// TIA Portal project "V15_PowerDistribution" (V15)

(* hardware
DEVICE "S7-1200 station_2"  S7-1200 Station
   slot 0: "Rack_0"  S7-1200 Rack  Rack  V1.0
   slot 1: "Main_PLC"  CPU 1214C DC/DC/DC  6ES7 214-1AG31-0XB0  V3.0
DEVICE "Main_HMI"  KTP700 Basic PN
   slot 0: "Main_HMI"  KTP700 Basic PN  6AV2 123-2GB03-0AX0  15.0.0.0
   slot 1: "HMI_RT_2"  KTP700 Basic PN  6AV2 123-2GB03-0AX0  15.0.0.0
   slot 5: "Main_HMI.IE_CP_1"  PROFINET Interface  15.0.0.0
      slot 1: "PROFINET Interface_1"  PROFINET Interface
         slot 1: "Port_1"  Port
DEVICE "S7-1200 station_1"  S7-1200 Station
   slot 0: "Rack_0"  S7-1200 Rack  Rack  V1.0
   slot 1: "Test_PLC"  CPU 1214C DC/DC/DC  6ES7 214-1AG40-0XB0  V4.2
DEVICE "Test_HMI"  KTP700 Basic PN
   slot 0: "Test_HMI"  KTP700 Basic PN  6AV2 123-2GB03-0AX0  15.0.0.0
   slot 1: "HMI_RT_1"  KTP700 Basic PN  6AV2 123-2GB03-0AX0  15.0.0.0
   slot 5: "Test_HMI.IE_CP_1"  PROFINET Interface  15.0.0.0
      slot 1: "PROFINET Interface_1"  PROFINET Interface
         slot 1: "Port_1"  Port
DEVICE "Main_PC"  SIMATIC PC station
   slot 0: "SIMATIC PC station"  Rail  SIMATIC PC-Station  V1.0
      slot 125: "Stationmanager"  Station_Manager  V6.0.4
   slot 1: "PC_HMI"  WinCC RT Advanced  6AV2 104-0xxxx-xxxx  15.0.0.0
      slot 33792: "Host interface"  Host interface
   slot 2: "IE general_1"  IE General  IE_CP  V8.2.0
*)

// ===== PLC "Main_PLC"  CPU 1214C DC/DC/DC =====

VAR_GLOBAL   // PLC tag table "Default tag table"
   "Clock_Byte" AT %MB0 : Byte;
   "Clock_10Hz" AT %M0.0 : Bool;
   "Clock_5Hz" AT %M0.1 : Bool;
   "Clock_2.5Hz" AT %M0.2 : Bool;
   "Clock_2Hz" AT %M0.3 : Bool;
   "Clock_1.25Hz" AT %M0.4 : Bool;
   "Clock_1Hz" AT %M0.5 : Bool;
   "Clock_0.625Hz" AT %M0.6 : Bool;
   "Clock_0.5Hz" AT %M0.7 : Bool;
   "Normal" AT %Q0.0 : Bool;
   "Low_Volt" AT %Q0.1 : Bool;
   "Short_Circuit" AT %Q0.2 : Bool;
   "Freq_Fault" AT %Q0.3 : Bool;
   "Open_Circuit" AT %Q0.4 : Bool;
   "Overload" AT %Q0.5 : Bool;
   "illegal_load" AT %Q0.6 : Bool;
   "Poor_PF" AT %Q0.7 : Bool;
   "CB" AT %Q1.1 : Bool;
   "Switch_auto" AT %M2.1 : Bool;
   "Switch_manual" AT %M1.0 : Bool;
   "Timer0_enable" AT %M1.1 : Bool;
END_VAR

VAR_GLOBAL   // PLC tag table "HOLD_REG"
   "Send_Frequency" AT %MW100 : Word;   // Send_Frequency
   "Send_Voltage" AT %MW102 : Word;   // Send_Voltage
   "Send_Current" AT %MW104 : Word;   // Send_Current
   "Send_EnergyHighByte" AT %MW106 : Word;   // Send_EnergyHighByte
   "Send_EnergyLowByte" AT %MW108 : Word;   // Send_EnergyLowByte
   "Send_ActivePower" AT %MW110 : Word;   // Send_ActivePower
   "Send_ReactivePower" AT %MW112 : Word;   // Send_ReactivePower
   "Send_PowerFactor" AT %MW114 : Word;   // Send_PowerFactor
   "Send_ActiveCounter" AT %MW118 : Word;   // Send_ActiveCounter
   "Recv_Frequency" AT %MW120 : Word;   // Recv_Frequency
   "Recv_Voltage" AT %MW122 : Word;   // Recv_Voltage
   "Recv_Current" AT %MW124 : Word;   // Recv_Current
   "Recv_EnergyHighByte" AT %MW126 : Word;   // Recv_EnergyHighByte
   "Recv_EnergyLowByte" AT %MW128 : Word;   // Recv_EnergyLowByte
   "Recv_ActivePower" AT %MW130 : Word;   // Recv_ActivePower
   "Recv_ReactivePower" AT %MW132 : Word;   // Recv_ReactivePower
   "Recv_PowerFactor" AT %MW134 : Word;   // Recv_PowerFactor
   "Recv_ErrorFlag" AT %MW136 : Word;   // Recv_ErrorFlag
   "Recv_ActiveCounter" AT %MW138 : Word;   // Recv_ActiveCounter
   "Send_ErrorFlag" AT %MW116 : Word;   // Send_ErrorFlag
END_VAR

DATA_BLOCK "Input_DB"   // DB1
{ S7_Optimized_Access := 'TRUE' }
VERSION : 0.1
   VAR
      "Send_Frequency [Hz]" : DInt := 0;
      "Send_Voltage [V]" : DInt := 0;
      "Send_Current [A]" : DInt := 0;
      "Send_Energy [KWh]" : DInt;
      "Send_ActivePwr [W]" : DInt := 0;
      "Send_ReactivePwr [KVAr]" : DInt;
      Send_PwrFactor : DInt := 0;
      "Recv_Frequency [Hz]" : DInt := 0;
      "Recv_Voltage [V]" : DInt := 0;
      "Recv_Current [A]" : DInt := 0;
      "Recv_Energy [KWh]" : DInt;
      "Recv_ActivePwr [W]" : DInt := 0;
      "Recv_ReactivePwr [KVAr]" : DInt;
      Recv_PwrFactor : DInt := 0;
      Send_Error : DInt;
      Recv_Error : DInt;
      Send_ActiveCounter : DInt;
      Recv_ActiveCounter : DInt;
   END_VAR
BEGIN
END_DATA_BLOCK

DATA_BLOCK "MB_Server_Data"   // DB2
{ S7_Optimized_Access := 'TRUE' }
VERSION : 0.1
   VAR
      CONNECT_ID : UInt := 2;
      IP_PORT : UInt := 502;
      NDR : Bool;
      DR : Bool;
      ERROR : Bool;
      STATUS : Word;
   END_VAR
BEGIN
END_DATA_BLOCK

DATA_BLOCK "Cond_DB"   // DB3
{ S7_Optimized_Access := 'TRUE' }
VERSION : 0.1
   VAR
      Recv_PwrLimit : DInt := 1000;
      error_ActivePwr : DInt;
      Psend_10percent : DInt;
      PwrFactor_Limit : DInt := 500;
      Freq_LowerLImit : DInt := 4750;
      Freq_UpperLimit : DInt := 5250;
      Current_Limit : DInt := 2;
      Vsend_limit_5percent : DInt := 2200;
      Vsend_limit_10percent : DInt := 2080;
      Vsend_High : DInt := 2420;
   END_VAR
BEGIN
END_DATA_BLOCK

DATA_BLOCK "MB_Client_Data"   // DB5
{ S7_Optimized_Access := 'TRUE' }
VERSION : 0.1
   VAR
      DISCONNECT : Bool;
      CONNECT_ID : UInt := 1;
      IP_ADDRESS : Array[0..3] of Byte;
      IP_PORT : UInt := 502;
      MB_MODE : USInt := 1;
      DATA_ADDRESS : UDInt := 0;
      DATA_LEN : UInt := 20;
      DONE : Bool;
      BUSY : Bool;
      ERROR : Bool;
      STATUS : Word;
   END_VAR
BEGIN
   IP_ADDRESS[0] := 192;
   IP_ADDRESS[1] := 168;
   IP_ADDRESS[2] := 0;
   IP_ADDRESS[3] := 103;
END_DATA_BLOCK

DATA_BLOCK "Fault_DB"   // DB6
{ S7_Optimized_Access := 'TRUE' }
VERSION : 0.1
   VAR
      None : Bool;
      Low_Voltage : Bool;
      Short_Circuit : Bool;
      Freq_fault : Bool;
      Open_Circuit : Bool;
      High_Voltage : Bool;
      Overload : Bool;
      Illegal_Load : Bool;
      Poor_PF : Bool;
   END_VAR
BEGIN
END_DATA_BLOCK

// folder: System blocks/Program resources

DATA_BLOCK "IEC_Timer_0_DB"   // DB7
{ S7_Optimized_Access := 'TRUE' }
AUTHOR : Simatic
FAMILY : IEC
NAME : IEC_TMR
VERSION : 1.0
// stored: InstanceOfName IEC_TIMER
"IEC_TIMER"
BEGIN
END_DATA_BLOCK

DATA_BLOCK "IEC_Timer_0_DB_1"   // DB9
{ S7_Optimized_Access := 'TRUE' }
AUTHOR : Simatic
FAMILY : IEC
NAME : IEC_TMR
VERSION : 1.0
// stored: InstanceOfName IEC_TIMER
"IEC_TIMER"
BEGIN
END_DATA_BLOCK

DATA_BLOCK "IEC_Timer_0_DB_2"   // DB10
{ S7_Optimized_Access := 'TRUE' }
AUTHOR : Simatic
FAMILY : IEC
NAME : IEC_TMR
VERSION : 1.0
// stored: InstanceOfName IEC_TIMER
"IEC_TIMER"
BEGIN
END_DATA_BLOCK

DATA_BLOCK "IEC_Timer_0_DB_3"   // DB11
{ S7_Optimized_Access := 'TRUE' }
AUTHOR : Simatic
FAMILY : IEC
NAME : IEC_TMR
VERSION : 1.0
// stored: InstanceOfName IEC_TIMER
"IEC_TIMER"
BEGIN
END_DATA_BLOCK

// folder: (top level)

ORGANIZATION_BLOCK "Main"   // OB1, LAD, ProgramCycle
TITLE = "Main Program Sweep (Cycle)"
{ S7_Optimized_Access := 'TRUE' }
VERSION : 0.1
   VAR_INPUT
      Initial_Call : Bool;   // Initial call of this OB
      Remanence : Bool;   // =True, if remanent data are available
   END_VAR
   VAR_TEMP
      Freq_Fault : Bool;
   END_VAR
BEGIN

REGION Network 1: Detect Fault
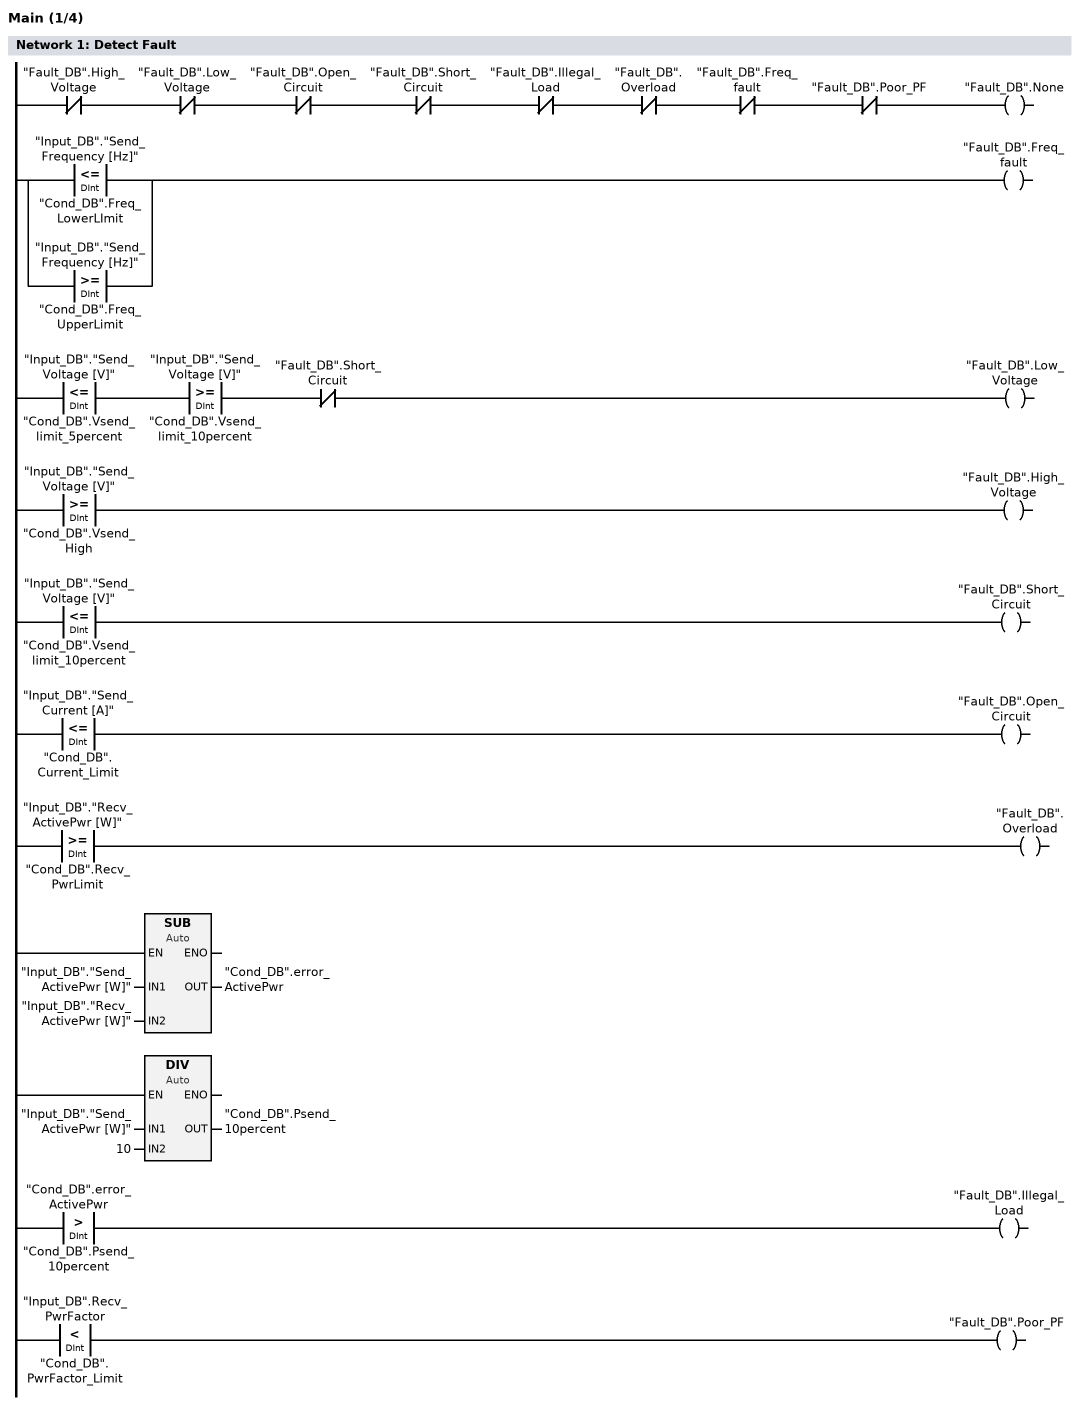
   RUNG wire#powerrail
      I_Contact( "Fault_DB".High_Voltage )
      I_Contact( "Fault_DB".Low_Voltage )
      I_Contact( "Fault_DB".Open_Circuit )
      I_Contact( "Fault_DB".Short_Circuit )
      I_Contact( "Fault_DB".Illegal_Load )
      I_Contact( "Fault_DB".Overload )
      I_Contact( "Fault_DB".Freq_fault )
      I_Contact( "Fault_DB".Poor_PF )
      Coil( "Fault_DB".None )
   END_RUNG
   RUNG wire#powerrail
      { S7_Templates := "SrcType := DInt" } LE_Contact(in1 := "Input_DB"."Send_Frequency [Hz]", in2 := "Cond_DB".Freq_LowerLImit)
      wire#w1
      Coil( "Fault_DB".Freq_fault )
   END_RUNG
   RUNG wire#powerrail
      { S7_Templates := "SrcType := DInt" } GE_Contact(in1 := "Input_DB"."Send_Frequency [Hz]", in2 := "Cond_DB".Freq_UpperLimit)
   END_RUNG wire#w1
   RUNG wire#powerrail
      { S7_Templates := "SrcType := DInt" } LE_Contact(in1 := "Input_DB"."Send_Voltage [V]", in2 := "Cond_DB".Vsend_limit_5percent)
      { S7_Templates := "SrcType := DInt" } GE_Contact(in1 := "Input_DB"."Send_Voltage [V]", in2 := "Cond_DB".Vsend_limit_10percent)
      I_Contact( "Fault_DB".Short_Circuit )
      Coil( "Fault_DB".Low_Voltage )
   END_RUNG
   RUNG wire#powerrail
      { S7_Templates := "SrcType := DInt" } GE_Contact(in1 := "Input_DB"."Send_Voltage [V]", in2 := "Cond_DB".Vsend_High)
      Coil( "Fault_DB".High_Voltage )
   END_RUNG
   RUNG wire#powerrail
      { S7_Templates := "SrcType := DInt" } LE_Contact(in1 := "Input_DB"."Send_Voltage [V]", in2 := "Cond_DB".Vsend_limit_10percent)
      Coil( "Fault_DB".Short_Circuit )
   END_RUNG
   RUNG wire#powerrail
      { S7_Templates := "SrcType := DInt" } LE_Contact(in1 := "Input_DB"."Send_Current [A]", in2 := "Cond_DB".Current_Limit)
      Coil( "Fault_DB".Open_Circuit )
   END_RUNG
   RUNG wire#powerrail
      { S7_Templates := "SrcType := DInt" } GE_Contact(in1 := "Input_DB"."Recv_ActivePwr [W]", in2 := "Cond_DB".Recv_PwrLimit)
      Coil( "Fault_DB".Overload )
   END_RUNG
   RUNG wire#powerrail
      { S7_GenerateENO := "TRUE" } Sub(in1 := "Input_DB"."Send_ActivePwr [W]", in2 := "Input_DB"."Recv_ActivePwr [W]", out => "Cond_DB".error_ActivePwr)
   END_RUNG
   RUNG wire#powerrail
      { S7_GenerateENO := "TRUE" } Div(in1 := "Input_DB"."Send_ActivePwr [W]", in2 := 10, out => "Cond_DB".Psend_10percent)
   END_RUNG
   RUNG wire#powerrail
      { S7_Templates := "SrcType := DInt" } GT_Contact(in1 := "Cond_DB".error_ActivePwr, in2 := "Cond_DB".Psend_10percent)
      Coil( "Fault_DB".Illegal_Load )
   END_RUNG
   RUNG wire#powerrail
      { S7_Templates := "SrcType := DInt" } LT_Contact(in1 := "Input_DB".Recv_PwrFactor, in2 := "Cond_DB".PwrFactor_Limit)
      Coil( "Fault_DB".Poor_PF )
   END_RUNG
   // the same network as SCL:
   "Fault_DB".None := NOT "Fault_DB".High_Voltage AND NOT "Fault_DB".Low_Voltage AND NOT "Fault_DB".Open_Circuit AND NOT "Fault_DB".Short_Circuit AND NOT "Fault_DB".Illegal_Load AND NOT "Fault_DB".Overload AND NOT "Fault_DB".Freq_fault AND NOT "Fault_DB".Poor_PF;
   "Fault_DB".Freq_fault := ("Input_DB"."Send_Frequency [Hz]" <= "Cond_DB".Freq_LowerLImit) OR ("Input_DB"."Send_Frequency [Hz]" >= "Cond_DB".Freq_UpperLimit);
   "Fault_DB".Low_Voltage := ("Input_DB"."Send_Voltage [V]" <= "Cond_DB".Vsend_limit_5percent) AND ("Input_DB"."Send_Voltage [V]" >= "Cond_DB".Vsend_limit_10percent) AND NOT "Fault_DB".Short_Circuit;
   "Fault_DB".High_Voltage := "Input_DB"."Send_Voltage [V]" >= "Cond_DB".Vsend_High;
   "Fault_DB".Short_Circuit := "Input_DB"."Send_Voltage [V]" <= "Cond_DB".Vsend_limit_10percent;
   "Fault_DB".Open_Circuit := "Input_DB"."Send_Current [A]" <= "Cond_DB".Current_Limit;
   "Fault_DB".Overload := "Input_DB"."Recv_ActivePwr [W]" >= "Cond_DB".Recv_PwrLimit;
   "Cond_DB".error_ActivePwr := "Input_DB"."Send_ActivePwr [W]" - "Input_DB"."Recv_ActivePwr [W]";
   "Cond_DB".Psend_10percent := "Input_DB"."Send_ActivePwr [W]" / 10;
   "Fault_DB".Illegal_Load := "Cond_DB".error_ActivePwr > "Cond_DB".Psend_10percent;
   "Fault_DB".Poor_PF := "Input_DB".Recv_PwrFactor < "Cond_DB".PwrFactor_Limit;
END_REGION

REGION Network 2: Display Fault
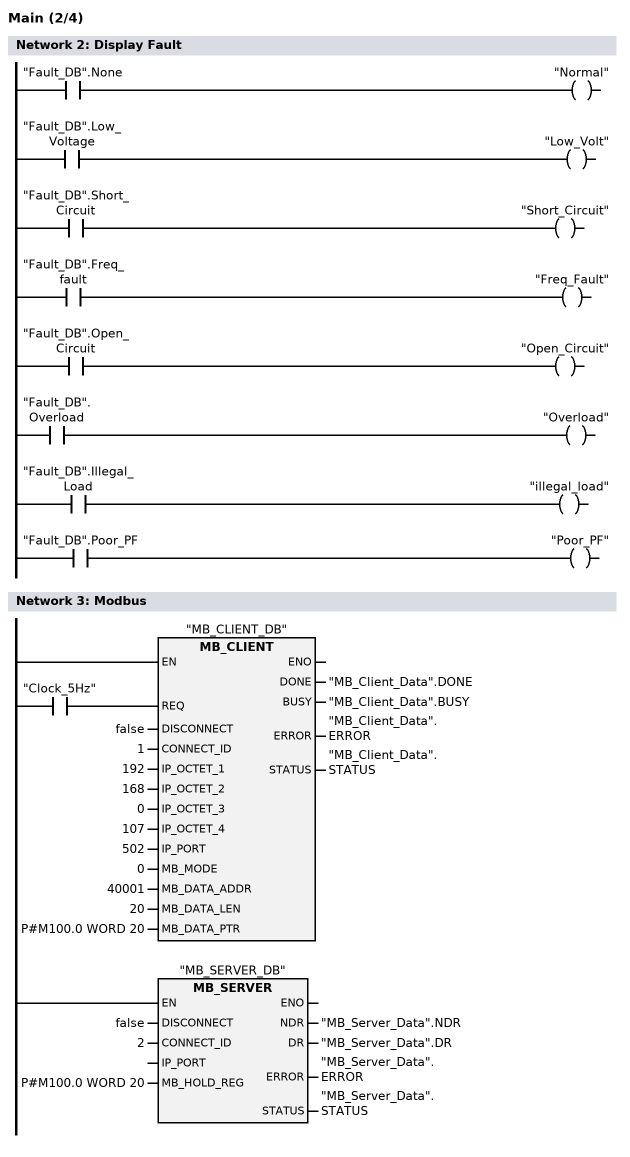
   RUNG wire#powerrail
      Contact( "Fault_DB".None )
      Coil( "Normal" )
   END_RUNG
   RUNG wire#powerrail
      Contact( "Fault_DB".Low_Voltage )
      Coil( "Low_Volt" )
   END_RUNG
   RUNG wire#powerrail
      Contact( "Fault_DB".Short_Circuit )
      Coil( "Short_Circuit" )
   END_RUNG
   RUNG wire#powerrail
      Contact( "Fault_DB".Freq_fault )
      Coil( "Freq_Fault" )
   END_RUNG
   RUNG wire#powerrail
      Contact( "Fault_DB".Open_Circuit )
      Coil( "Open_Circuit" )
   END_RUNG
   RUNG wire#powerrail
      Contact( "Fault_DB".Overload )
      Coil( "Overload" )
   END_RUNG
   RUNG wire#powerrail
      Contact( "Fault_DB".Illegal_Load )
      Coil( "illegal_load" )
   END_RUNG
   RUNG wire#powerrail
      Contact( "Fault_DB".Poor_PF )
      Coil( "Poor_PF" )
   END_RUNG
   // the same network as SCL:
   "Normal" := "Fault_DB".None;
   "Low_Volt" := "Fault_DB".Low_Voltage;
   "Short_Circuit" := "Fault_DB".Short_Circuit;
   "Freq_Fault" := "Fault_DB".Freq_fault;
   "Open_Circuit" := "Fault_DB".Open_Circuit;
   "Overload" := "Fault_DB".Overload;
   "illegal_load" := "Fault_DB".Illegal_Load;
   "Poor_PF" := "Fault_DB".Poor_PF;
END_REGION

REGION Network 3: Modbus
   "MB_CLIENT_DB"(REQ := "Clock_5Hz",   // MB_CLIENT
                  DISCONNECT := false,
                  CONNECT_ID := 1,
                  IP_OCTET_1 := 192,
                  IP_OCTET_2 := 168,
                  IP_OCTET_3 := 0,
                  IP_OCTET_4 := 107,
                  IP_PORT := 502,
                  MB_MODE := 0,
                  MB_DATA_ADDR := 40001,
                  MB_DATA_LEN := 20,
                  MB_DATA_PTR := P#M100.0 WORD 20,
                  DONE => "MB_Client_Data".DONE,
                  BUSY => "MB_Client_Data".BUSY,
                  ERROR => "MB_Client_Data".ERROR,
                  STATUS => "MB_Client_Data".STATUS);
   "MB_SERVER_DB"(DISCONNECT := false,   // MB_SERVER
                  CONNECT_ID := 2,
                  MB_HOLD_REG := P#M100.0 WORD 20,
                  NDR => "MB_Server_Data".NDR,
                  DR => "MB_Server_Data".DR,
                  ERROR => "MB_Server_Data".ERROR,
                  STATUS => "MB_Server_Data".STATUS);
END_REGION

REGION Network 4: Map data from sensors to DB
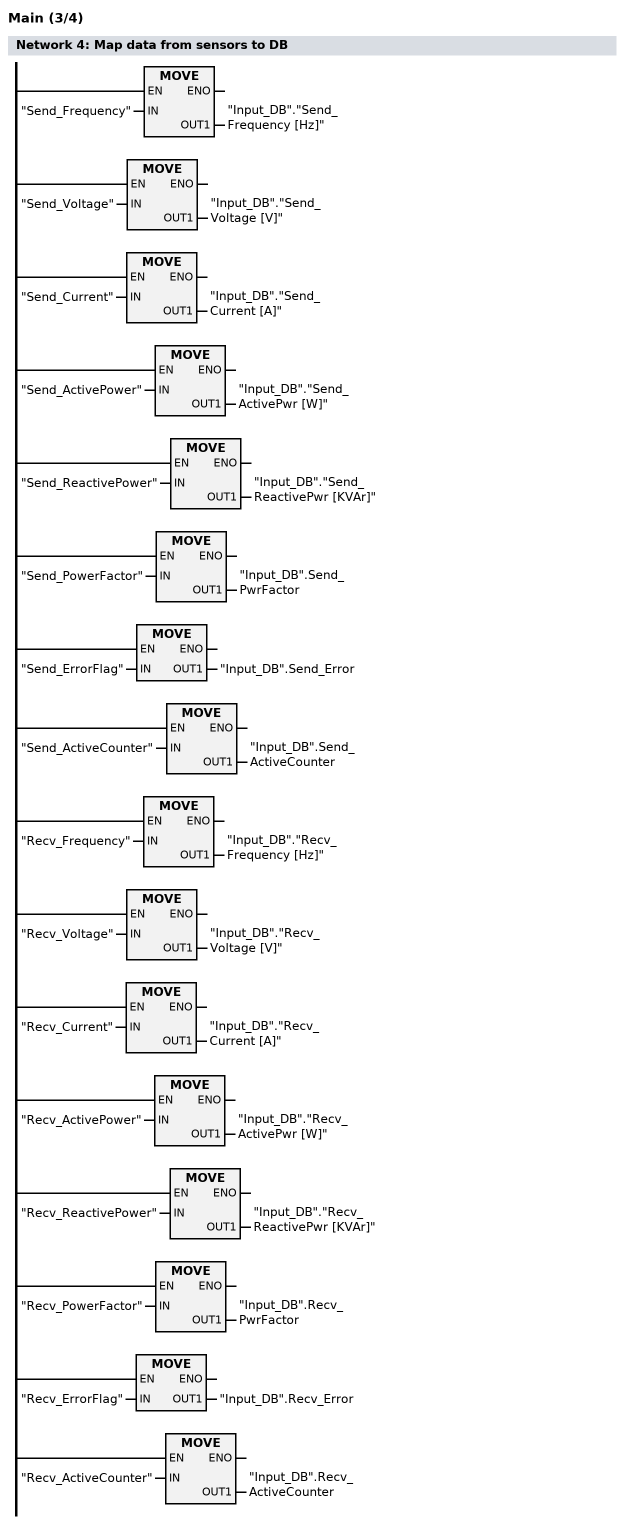
   RUNG wire#powerrail
      { S7_GenerateENO := "TRUE" } Move(in := "Send_Frequency", out1 => "Input_DB"."Send_Frequency [Hz]")
   END_RUNG
   RUNG wire#powerrail
      { S7_GenerateENO := "TRUE" } Move(in := "Send_Voltage", out1 => "Input_DB"."Send_Voltage [V]")
   END_RUNG
   RUNG wire#powerrail
      { S7_GenerateENO := "TRUE" } Move(in := "Send_Current", out1 => "Input_DB"."Send_Current [A]")
   END_RUNG
   RUNG wire#powerrail
      { S7_GenerateENO := "TRUE" } Move(in := "Send_ActivePower", out1 => "Input_DB"."Send_ActivePwr [W]")
   END_RUNG
   RUNG wire#powerrail
      { S7_GenerateENO := "TRUE" } Move(in := "Send_ReactivePower", out1 => "Input_DB"."Send_ReactivePwr [KVAr]")
   END_RUNG
   RUNG wire#powerrail
      { S7_GenerateENO := "TRUE" } Move(in := "Send_PowerFactor", out1 => "Input_DB".Send_PwrFactor)
   END_RUNG
   RUNG wire#powerrail
      { S7_GenerateENO := "TRUE" } Move(in := "Send_ErrorFlag", out1 => "Input_DB".Send_Error)
   END_RUNG
   RUNG wire#powerrail
      { S7_GenerateENO := "TRUE" } Move(in := "Send_ActiveCounter", out1 => "Input_DB".Send_ActiveCounter)
   END_RUNG
   RUNG wire#powerrail
      { S7_GenerateENO := "TRUE" } Move(in := "Recv_Frequency", out1 => "Input_DB"."Recv_Frequency [Hz]")
   END_RUNG
   RUNG wire#powerrail
      { S7_GenerateENO := "TRUE" } Move(in := "Recv_Voltage", out1 => "Input_DB"."Recv_Voltage [V]")
   END_RUNG
   RUNG wire#powerrail
      { S7_GenerateENO := "TRUE" } Move(in := "Recv_Current", out1 => "Input_DB"."Recv_Current [A]")
   END_RUNG
   RUNG wire#powerrail
      { S7_GenerateENO := "TRUE" } Move(in := "Recv_ActivePower", out1 => "Input_DB"."Recv_ActivePwr [W]")
   END_RUNG
   RUNG wire#powerrail
      { S7_GenerateENO := "TRUE" } Move(in := "Recv_ReactivePower", out1 => "Input_DB"."Recv_ReactivePwr [KVAr]")
   END_RUNG
   RUNG wire#powerrail
      { S7_GenerateENO := "TRUE" } Move(in := "Recv_PowerFactor", out1 => "Input_DB".Recv_PwrFactor)
   END_RUNG
   RUNG wire#powerrail
      { S7_GenerateENO := "TRUE" } Move(in := "Recv_ErrorFlag", out1 => "Input_DB".Recv_Error)
   END_RUNG
   RUNG wire#powerrail
      { S7_GenerateENO := "TRUE" } Move(in := "Recv_ActiveCounter", out1 => "Input_DB".Recv_ActiveCounter)
   END_RUNG
   // the same network as SCL:
   "Input_DB"."Send_Frequency [Hz]" := "Send_Frequency";
   "Input_DB"."Send_Voltage [V]" := "Send_Voltage";
   "Input_DB"."Send_Current [A]" := "Send_Current";
   "Input_DB"."Send_ActivePwr [W]" := "Send_ActivePower";
   "Input_DB"."Send_ReactivePwr [KVAr]" := "Send_ReactivePower";
   "Input_DB".Send_PwrFactor := "Send_PowerFactor";
   "Input_DB".Send_Error := "Send_ErrorFlag";
   "Input_DB".Send_ActiveCounter := "Send_ActiveCounter";
   "Input_DB"."Recv_Frequency [Hz]" := "Recv_Frequency";
   "Input_DB"."Recv_Voltage [V]" := "Recv_Voltage";
   "Input_DB"."Recv_Current [A]" := "Recv_Current";
   "Input_DB"."Recv_ActivePwr [W]" := "Recv_ActivePower";
   "Input_DB"."Recv_ReactivePwr [KVAr]" := "Recv_ReactivePower";
   "Input_DB".Recv_PwrFactor := "Recv_PowerFactor";
   "Input_DB".Recv_Error := "Recv_ErrorFlag";
   "Input_DB".Recv_ActiveCounter := "Recv_ActiveCounter";
END_REGION

REGION Network 5: Circuit Breaker Switch
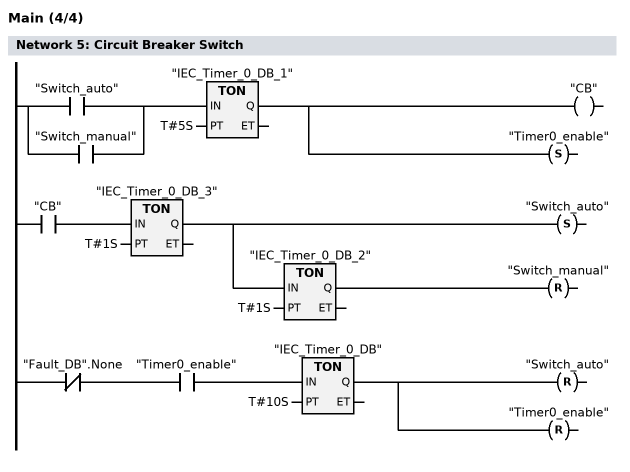
   "IEC_Timer_0_DB_1".TON(IN := "Switch_auto" OR "Switch_manual", PT := T#5S);
   "CB" := "IEC_Timer_0_DB_1".Q;
   IF "IEC_Timer_0_DB_1".Q THEN "Timer0_enable" := TRUE; END_IF;
   "IEC_Timer_0_DB_3".TON(IN := "CB", PT := T#1S);
   IF "IEC_Timer_0_DB_3".Q THEN "Switch_auto" := TRUE; END_IF;
   "IEC_Timer_0_DB_2".TON(IN := "IEC_Timer_0_DB_3".Q, PT := T#1S);
   IF "IEC_Timer_0_DB_2".Q THEN "Switch_manual" := FALSE; END_IF;
   "IEC_Timer_0_DB".TON(IN := NOT "Fault_DB".None AND "Timer0_enable", PT := T#10S);
   IF "IEC_Timer_0_DB".Q THEN
       "Switch_auto" := FALSE;
       "Timer0_enable" := FALSE;
   END_IF;
END_REGION
END_ORGANIZATION_BLOCK

// ===== PLC "Test_PLC"  CPU 1214C DC/DC/DC =====

VAR_GLOBAL   // PLC tag table "Default tag table"
   "Clock_Byte" AT %MB0 : Byte;
   "Clock_10Hz" AT %M0.0 : Bool;
   "Clock_5Hz" AT %M0.1 : Bool;
   "Clock_2.5Hz" AT %M0.2 : Bool;
   "Clock_2Hz" AT %M0.3 : Bool;
   "Clock_1.25Hz" AT %M0.4 : Bool;
   "Clock_1Hz" AT %M0.5 : Bool;
   "Clock_0.625Hz" AT %M0.6 : Bool;
   "Clock_0.5Hz" AT %M0.7 : Bool;
   "Normal" AT %M1.0 : Bool;
   "Low_Volt" AT %M1.1 : Bool;
   "Short_Circuit" AT %M1.2 : Bool;
   "Freq_Fault" AT %M1.3 : Bool;
   "Open_Circuit" AT %M1.4 : Bool;
   "Overload" AT %M1.5 : Bool;
   "illegal_load" AT %M1.6 : Bool;
   "Poor_PF" AT %M1.7 : Bool;
   "CB" AT %M2.0 : Bool;
   "CB_enable" AT %M2.1 : Bool;
END_VAR

VAR_GLOBAL   // PLC tag table "HOLD_REG"
   "40001" AT %MW100 : Word;   // Send_Frequency
   "40002" AT %MW102 : Word;   // Send_Voltage
   "40003" AT %MW104 : Word;   // Send_Current
   "40004" AT %MW106 : Word;   // Send_EnergyHighByte
   "40005" AT %MW108 : Word;   // Send_EnergyLowByte
   "40006" AT %MW110 : Word;   // Send_ActivePower
   "40007" AT %MW112 : Word;   // Send_ReactivePower
   "40008" AT %MW114 : Word;   // Send_PowerFactor
   "40009" AT %MW116 : Word;   // Recv_Frequency
   "40010" AT %MW118 : Word;   // Recv_Voltage
   "40011" AT %MW120 : Word;   // Recv_Current
   "40012" AT %MW122 : Word;   // Recv_EnergyHighByte
   "40013" AT %MW124 : Word;   // Recv_EnergyLowByte
   "40014" AT %MW126 : Word;   // Recv_ActivePower
   "40015" AT %MW128 : Word;   // Recv_ReactivePower
   "40016" AT %MW130 : Word;   // Recv_PowerFactor
   "40017" AT %MW132 : Word;   // Send_ErrorFlag
   "40018" AT %MW134 : Word;   // Recv_ErrorFlag
   "40019" AT %MW136 : Word;   // Send_ActiveCounter
   "40020" AT %MW138 : Word;   // Recv_ActiveCounter
END_VAR

DATA_BLOCK "Input_DB"   // DB1
{ S7_Optimized_Access := 'TRUE' }
VERSION : 0.1
   VAR
      "Send_Frequency [Hz]" : DInt := 0;
      "Send_Voltage [V]" : DInt := 0;
      "Send_Current [mA]" : DInt := 0;
      "Send_Energy [KWh]" : DInt;
      "Send_ActivePwr [W]" : DInt := 0;
      "Send_ReactivePwr [KVAr]" : DInt;
      Send_PwrFactor : DInt := 0;
      "Recv_Frequency [Hz]" : DInt := 0;
      "Recv_Voltage [V]" : DInt := 0;
      "Recv_Current [mA]" : DInt := 0;
      "Recv_Energy [KWh]" : DInt;
      "Recv_ActivePwr [W]" : DInt := 0;
      "Recv_ReactivePwr [KVAr]" : DInt;
      Recv_PwrFactor : DInt := 0;
      Send_Error : DInt;
      Recv_Error : DInt;
      Send_ActiveCounter : DInt;
      Recv_ActiveCounter : DInt;
   END_VAR
BEGIN
END_DATA_BLOCK

DATA_BLOCK "Fault_DB"   // DB2
{ S7_Optimized_Access := 'TRUE' }
VERSION : 0.1
   VAR
      None : Bool;
      Low_Voltage : Bool;
      Short_Circuit : Bool;
      Freq_fault : Bool;
      Open_Circuit : Bool;
      High_Voltage : Bool;
      Overload : Bool;
      Illegal_Load : Bool;
      Poor_PF : Bool;
   END_VAR
BEGIN
END_DATA_BLOCK

DATA_BLOCK "Cond_DB"   // DB3
{ S7_Optimized_Access := 'TRUE' }
VERSION : 0.1
   VAR
      Recv_PwrLimit : DInt := 1000;
      error_ActivePwr : DInt;
      Psend_10percent : DInt;
      PwrFactor_Limit : DInt := 800;
      Freq_LowerLImit : DInt := 4750;
      Freq_UpperLimit : DInt := 5250;
      Current_Limit : DInt := 2;
      Vsend_limit_5percent : DInt := 2200;
      Vsend_limit_10percent : DInt := 2080;
      Vsend_High : DInt := 2420;
   END_VAR
BEGIN
END_DATA_BLOCK

DATA_BLOCK "MB_Client_Data"   // DB5
{ S7_Optimized_Access := 'TRUE' }
VERSION : 0.1
   VAR
      DISCONNECT : Bool;
      CONNECT_ID : UInt := 1;
      IP_ADDRESS : Array[0..3] of Byte;
      IP_PORT : UInt := 502;
      MB_MODE : USInt := 1;
      DATA_ADDRESS : UDInt := 0;
      DATA_LEN : UInt := 20;
      DONE : Bool;
      BUSY : Bool;
      ERROR : Bool;
      STATUS : Word;
   END_VAR
BEGIN
   IP_ADDRESS[0] := 192;
   IP_ADDRESS[1] := 168;
   IP_ADDRESS[2] := 0;
   IP_ADDRESS[3] := 103;
END_DATA_BLOCK

ORGANIZATION_BLOCK "Main"   // OB1, LAD, ProgramCycle
TITLE = "Main Program Sweep (Cycle)"
{ S7_Optimized_Access := 'TRUE' }
VERSION : 0.1
   VAR_INPUT
      Initial_Call : Bool;   // Initial call of this OB
      Remanence : Bool;   // =True, if remanent data are available
   END_VAR
   VAR_TEMP
      Freq_Fault : Bool;
   END_VAR
BEGIN

REGION Network 1: Detect Fault
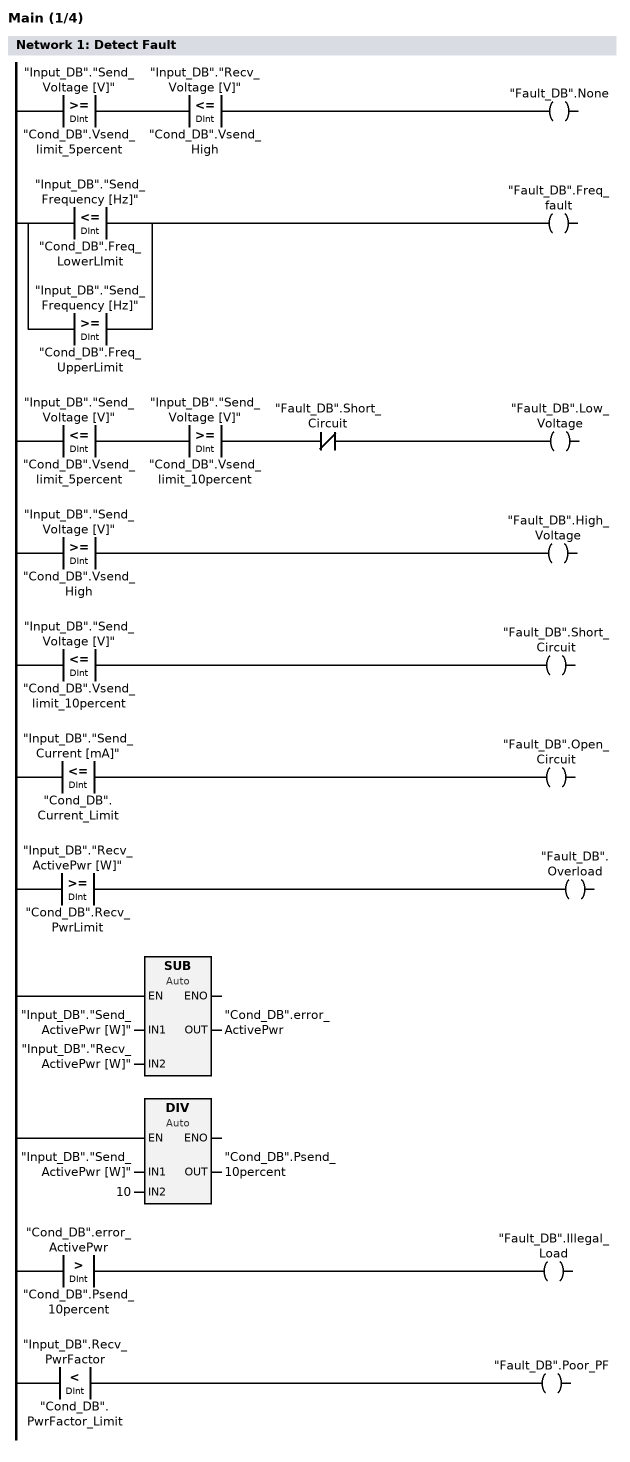
   RUNG wire#powerrail
      { S7_Templates := "SrcType := DInt" } GE_Contact(in1 := "Input_DB"."Send_Voltage [V]", in2 := "Cond_DB".Vsend_limit_5percent)
      { S7_Templates := "SrcType := DInt" } LE_Contact(in1 := "Input_DB"."Recv_Voltage [V]", in2 := "Cond_DB".Vsend_High)
      Coil( "Fault_DB".None )
   END_RUNG
   RUNG wire#powerrail
      { S7_Templates := "SrcType := DInt" } LE_Contact(in1 := "Input_DB"."Send_Frequency [Hz]", in2 := "Cond_DB".Freq_LowerLImit)
      wire#w1
      Coil( "Fault_DB".Freq_fault )
   END_RUNG
   RUNG wire#powerrail
      { S7_Templates := "SrcType := DInt" } GE_Contact(in1 := "Input_DB"."Send_Frequency [Hz]", in2 := "Cond_DB".Freq_UpperLimit)
   END_RUNG wire#w1
   RUNG wire#powerrail
      { S7_Templates := "SrcType := DInt" } LE_Contact(in1 := "Input_DB"."Send_Voltage [V]", in2 := "Cond_DB".Vsend_limit_5percent)
      { S7_Templates := "SrcType := DInt" } GE_Contact(in1 := "Input_DB"."Send_Voltage [V]", in2 := "Cond_DB".Vsend_limit_10percent)
      I_Contact( "Fault_DB".Short_Circuit )
      Coil( "Fault_DB".Low_Voltage )
   END_RUNG
   RUNG wire#powerrail
      { S7_Templates := "SrcType := DInt" } GE_Contact(in1 := "Input_DB"."Send_Voltage [V]", in2 := "Cond_DB".Vsend_High)
      Coil( "Fault_DB".High_Voltage )
   END_RUNG
   RUNG wire#powerrail
      { S7_Templates := "SrcType := DInt" } LE_Contact(in1 := "Input_DB"."Send_Voltage [V]", in2 := "Cond_DB".Vsend_limit_10percent)
      Coil( "Fault_DB".Short_Circuit )
   END_RUNG
   RUNG wire#powerrail
      { S7_Templates := "SrcType := DInt" } LE_Contact(in1 := "Input_DB"."Send_Current [mA]", in2 := "Cond_DB".Current_Limit)
      Coil( "Fault_DB".Open_Circuit )
   END_RUNG
   RUNG wire#powerrail
      { S7_Templates := "SrcType := DInt" } GE_Contact(in1 := "Input_DB"."Recv_ActivePwr [W]", in2 := "Cond_DB".Recv_PwrLimit)
      Coil( "Fault_DB".Overload )
   END_RUNG
   RUNG wire#powerrail
      { S7_GenerateENO := "TRUE" } Sub(in1 := "Input_DB"."Send_ActivePwr [W]", in2 := "Input_DB"."Recv_ActivePwr [W]", out => "Cond_DB".error_ActivePwr)
   END_RUNG
   RUNG wire#powerrail
      { S7_GenerateENO := "TRUE" } Div(in1 := "Input_DB"."Send_ActivePwr [W]", in2 := 10, out => "Cond_DB".Psend_10percent)
   END_RUNG
   RUNG wire#powerrail
      { S7_Templates := "SrcType := DInt" } GT_Contact(in1 := "Cond_DB".error_ActivePwr, in2 := "Cond_DB".Psend_10percent)
      Coil( "Fault_DB".Illegal_Load )
   END_RUNG
   RUNG wire#powerrail
      { S7_Templates := "SrcType := DInt" } LT_Contact(in1 := "Input_DB".Recv_PwrFactor, in2 := "Cond_DB".PwrFactor_Limit)
      Coil( "Fault_DB".Poor_PF )
   END_RUNG
   // the same network as SCL:
   "Fault_DB".None := ("Input_DB"."Send_Voltage [V]" >= "Cond_DB".Vsend_limit_5percent) AND ("Input_DB"."Recv_Voltage [V]" <= "Cond_DB".Vsend_High);
   "Fault_DB".Freq_fault := ("Input_DB"."Send_Frequency [Hz]" <= "Cond_DB".Freq_LowerLImit) OR ("Input_DB"."Send_Frequency [Hz]" >= "Cond_DB".Freq_UpperLimit);
   "Fault_DB".Low_Voltage := ("Input_DB"."Send_Voltage [V]" <= "Cond_DB".Vsend_limit_5percent) AND ("Input_DB"."Send_Voltage [V]" >= "Cond_DB".Vsend_limit_10percent) AND NOT "Fault_DB".Short_Circuit;
   "Fault_DB".High_Voltage := "Input_DB"."Send_Voltage [V]" >= "Cond_DB".Vsend_High;
   "Fault_DB".Short_Circuit := "Input_DB"."Send_Voltage [V]" <= "Cond_DB".Vsend_limit_10percent;
   "Fault_DB".Open_Circuit := "Input_DB"."Send_Current [mA]" <= "Cond_DB".Current_Limit;
   "Fault_DB".Overload := "Input_DB"."Recv_ActivePwr [W]" >= "Cond_DB".Recv_PwrLimit;
   "Cond_DB".error_ActivePwr := "Input_DB"."Send_ActivePwr [W]" - "Input_DB"."Recv_ActivePwr [W]";
   "Cond_DB".Psend_10percent := "Input_DB"."Send_ActivePwr [W]" / 10;
   "Fault_DB".Illegal_Load := "Cond_DB".error_ActivePwr > "Cond_DB".Psend_10percent;
   "Fault_DB".Poor_PF := "Input_DB".Recv_PwrFactor < "Cond_DB".PwrFactor_Limit;
END_REGION

REGION Network 2: Display Fault
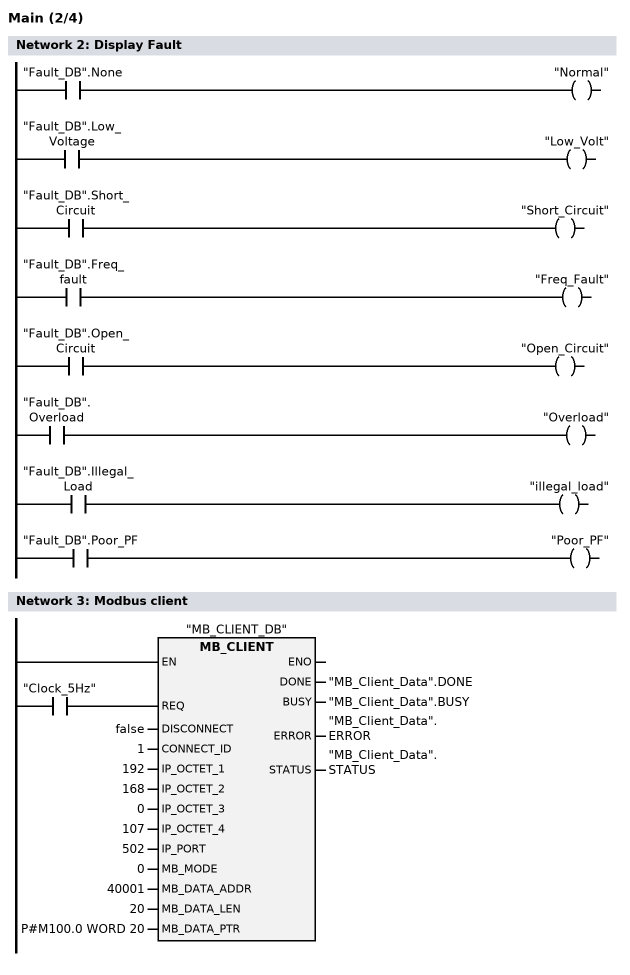
   RUNG wire#powerrail
      Contact( "Fault_DB".None )
      Coil( "Normal" )
   END_RUNG
   RUNG wire#powerrail
      Contact( "Fault_DB".Low_Voltage )
      Coil( "Low_Volt" )
   END_RUNG
   RUNG wire#powerrail
      Contact( "Fault_DB".Short_Circuit )
      Coil( "Short_Circuit" )
   END_RUNG
   RUNG wire#powerrail
      Contact( "Fault_DB".Freq_fault )
      Coil( "Freq_Fault" )
   END_RUNG
   RUNG wire#powerrail
      Contact( "Fault_DB".Open_Circuit )
      Coil( "Open_Circuit" )
   END_RUNG
   RUNG wire#powerrail
      Contact( "Fault_DB".Overload )
      Coil( "Overload" )
   END_RUNG
   RUNG wire#powerrail
      Contact( "Fault_DB".Illegal_Load )
      Coil( "illegal_load" )
   END_RUNG
   RUNG wire#powerrail
      Contact( "Fault_DB".Poor_PF )
      Coil( "Poor_PF" )
   END_RUNG
   // the same network as SCL:
   "Normal" := "Fault_DB".None;
   "Low_Volt" := "Fault_DB".Low_Voltage;
   "Short_Circuit" := "Fault_DB".Short_Circuit;
   "Freq_Fault" := "Fault_DB".Freq_fault;
   "Open_Circuit" := "Fault_DB".Open_Circuit;
   "Overload" := "Fault_DB".Overload;
   "illegal_load" := "Fault_DB".Illegal_Load;
   "Poor_PF" := "Fault_DB".Poor_PF;
END_REGION

REGION Network 3: Modbus client
   "MB_CLIENT_DB"(REQ := "Clock_5Hz",   // MB_CLIENT
                  DISCONNECT := false,
                  CONNECT_ID := 1,
                  IP_OCTET_1 := 192,
                  IP_OCTET_2 := 168,
                  IP_OCTET_3 := 0,
                  IP_OCTET_4 := 107,
                  IP_PORT := 502,
                  MB_MODE := 0,
                  MB_DATA_ADDR := 40001,
                  MB_DATA_LEN := 20,
                  MB_DATA_PTR := P#M100.0 WORD 20,
                  DONE => "MB_Client_Data".DONE,
                  BUSY => "MB_Client_Data".BUSY,
                  ERROR => "MB_Client_Data".ERROR,
                  STATUS => "MB_Client_Data".STATUS);
END_REGION

REGION Network 4: Map data from sensors to DB
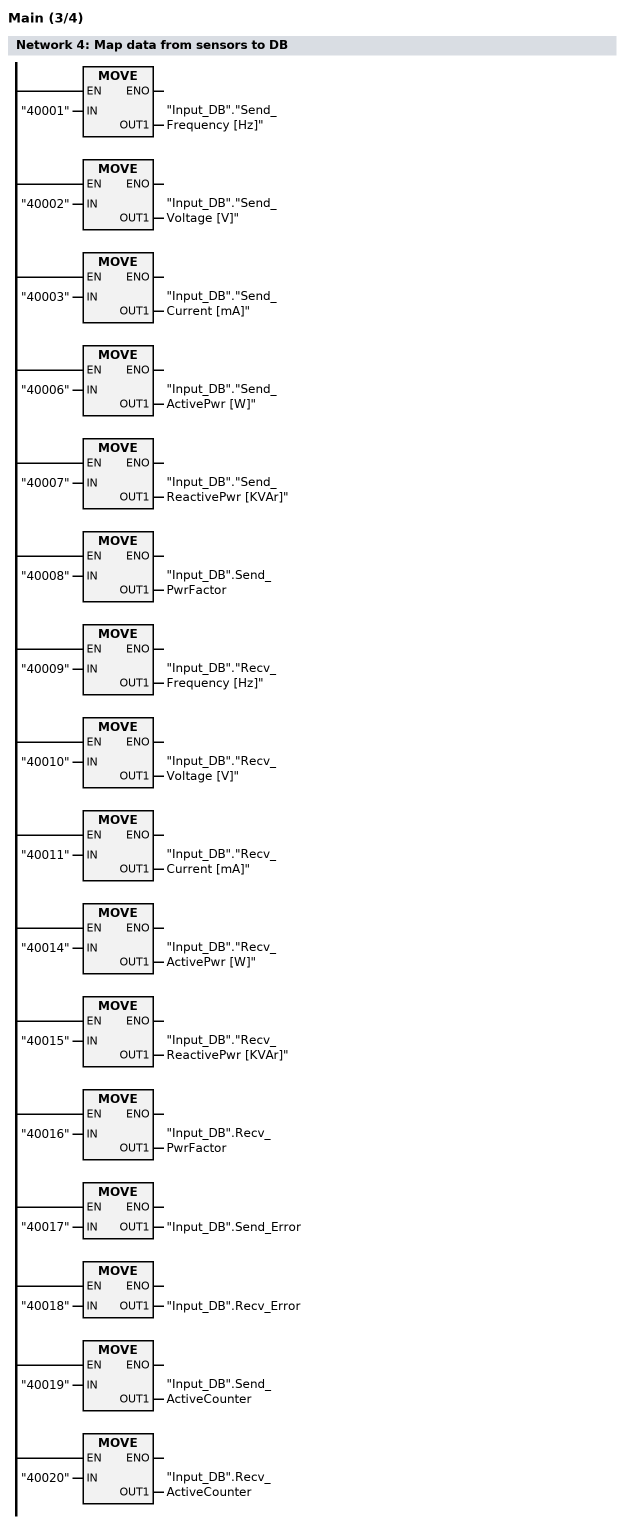
   RUNG wire#powerrail
      { S7_GenerateENO := "TRUE" } Move(in := "40001", out1 => "Input_DB"."Send_Frequency [Hz]")
   END_RUNG
   RUNG wire#powerrail
      { S7_GenerateENO := "TRUE" } Move(in := "40002", out1 => "Input_DB"."Send_Voltage [V]")
   END_RUNG
   RUNG wire#powerrail
      { S7_GenerateENO := "TRUE" } Move(in := "40003", out1 => "Input_DB"."Send_Current [mA]")
   END_RUNG
   RUNG wire#powerrail
      { S7_GenerateENO := "TRUE" } Move(in := "40006", out1 => "Input_DB"."Send_ActivePwr [W]")
   END_RUNG
   RUNG wire#powerrail
      { S7_GenerateENO := "TRUE" } Move(in := "40007", out1 => "Input_DB"."Send_ReactivePwr [KVAr]")
   END_RUNG
   RUNG wire#powerrail
      { S7_GenerateENO := "TRUE" } Move(in := "40008", out1 => "Input_DB".Send_PwrFactor)
   END_RUNG
   RUNG wire#powerrail
      { S7_GenerateENO := "TRUE" } Move(in := "40009", out1 => "Input_DB"."Recv_Frequency [Hz]")
   END_RUNG
   RUNG wire#powerrail
      { S7_GenerateENO := "TRUE" } Move(in := "40010", out1 => "Input_DB"."Recv_Voltage [V]")
   END_RUNG
   RUNG wire#powerrail
      { S7_GenerateENO := "TRUE" } Move(in := "40011", out1 => "Input_DB"."Recv_Current [mA]")
   END_RUNG
   RUNG wire#powerrail
      { S7_GenerateENO := "TRUE" } Move(in := "40014", out1 => "Input_DB"."Recv_ActivePwr [W]")
   END_RUNG
   RUNG wire#powerrail
      { S7_GenerateENO := "TRUE" } Move(in := "40015", out1 => "Input_DB"."Recv_ReactivePwr [KVAr]")
   END_RUNG
   RUNG wire#powerrail
      { S7_GenerateENO := "TRUE" } Move(in := "40016", out1 => "Input_DB".Recv_PwrFactor)
   END_RUNG
   RUNG wire#powerrail
      { S7_GenerateENO := "TRUE" } Move(in := "40017", out1 => "Input_DB".Send_Error)
   END_RUNG
   RUNG wire#powerrail
      { S7_GenerateENO := "TRUE" } Move(in := "40018", out1 => "Input_DB".Recv_Error)
   END_RUNG
   RUNG wire#powerrail
      { S7_GenerateENO := "TRUE" } Move(in := "40019", out1 => "Input_DB".Send_ActiveCounter)
   END_RUNG
   RUNG wire#powerrail
      { S7_GenerateENO := "TRUE" } Move(in := "40020", out1 => "Input_DB".Recv_ActiveCounter)
   END_RUNG
   // the same network as SCL:
   "Input_DB"."Send_Frequency [Hz]" := "40001";
   "Input_DB"."Send_Voltage [V]" := "40002";
   "Input_DB"."Send_Current [mA]" := "40003";
   "Input_DB"."Send_ActivePwr [W]" := "40006";
   "Input_DB"."Send_ReactivePwr [KVAr]" := "40007";
   "Input_DB".Send_PwrFactor := "40008";
   "Input_DB"."Recv_Frequency [Hz]" := "40009";
   "Input_DB"."Recv_Voltage [V]" := "40010";
   "Input_DB"."Recv_Current [mA]" := "40011";
   "Input_DB"."Recv_ActivePwr [W]" := "40014";
   "Input_DB"."Recv_ReactivePwr [KVAr]" := "40015";
   "Input_DB".Recv_PwrFactor := "40016";
   "Input_DB".Send_Error := "40017";
   "Input_DB".Recv_Error := "40018";
   "Input_DB".Send_ActiveCounter := "40019";
   "Input_DB".Recv_ActiveCounter := "40020";
END_REGION

REGION Network 5: Circuit Breaker Switch
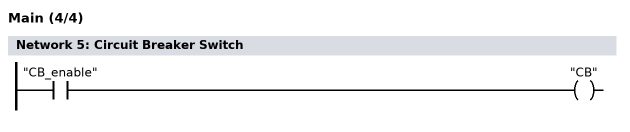
   RUNG wire#powerrail
      Contact( "CB_enable" )
      Coil( "CB" )
   END_RUNG
   // the same network as SCL:
   "CB" := "CB_enable";
END_REGION
END_ORGANIZATION_BLOCK

(* ===== HMI "HMI_RT_2" =====
system functions are stored by id; their names below are inferred from use
connection "Main_Conn": ETHERNET, SMART_S7_1200_OMS

HMI tags "Default tag table"
   "Fault_DB_Illegal_Load" : Bool = PLC Fault_DB.Illegal_Load, 1 s
   "Fault_DB_Low_Voltage" : Bool = PLC Fault_DB.Low_Voltage, 1 s
   "Fault_DB_Open_Circuit" : Bool = PLC Fault_DB.Open_Circuit, 1 s
   "Fault_DB_Overload" : Bool = PLC Fault_DB.Overload, 1 s
   "Fault_DB_Poor_PF" : Bool = PLC Fault_DB.Poor_PF, 1 s
   "Fault_DB_Short_Circuit" : Bool = PLC Fault_DB.Short_Circuit, 1 s
   "Fault_DB_None" : Bool = PLC Fault_DB.None, 1 s
   "Fault_DB_Freq_fault" : Bool = PLC Fault_DB.Freq_fault, 1 s
   "Input_DB_Send_Frequency [Hz]" : DInt = PLC Input_DB."Send_Frequency [Hz]", 1 s
   "Input_DB_Recv_Frequency [Hz]" : DInt = PLC Input_DB."Recv_Frequency [Hz]", 1 s
   "Input_DB_Send_Voltage [V]" : DInt = PLC Input_DB."Send_Voltage [V]", 1 s
   "Input_DB_Recv_Voltage [V]" : DInt = PLC Input_DB."Recv_Voltage [V]", 1 s
   "Input_DB_Send_Current [mA]" : DInt = PLC Input_DB."Send_Current [A]", 1 s
   "Input_DB_Recv_Current [mA]" : DInt = PLC Input_DB."Recv_Current [A]", 1 s
   "Input_DB_Send_ActivePwr [W]" : DInt = PLC Input_DB."Send_ActivePwr [W]", 1 s
   "Input_DB_Recv_ActivePwr [W]" : DInt = PLC Input_DB."Recv_ActivePwr [W]", 1 s
   "Input_DB_Send_PwrFactor" : DInt = PLC Input_DB.Send_PwrFactor, 1 s
   "Input_DB_Recv_PwrFactor" : DInt = PLC Input_DB.Recv_PwrFactor, 1 s
   "Input_DB_Send_Error" : DInt = PLC Input_DB.Send_Error, 1 s
   "Input_DB_Recv_Error" : DInt = PLC Input_DB.Recv_Error, 1 s
   "CB_enable" : Bool = PLC Switch_auto AT %M2.1, 1 s
   "Switch_manual" : Bool = PLC Switch_manual AT %M1.0, 1 s

Template "Template_1" 800x480
   Button "Exit" at 714,429 size 71x50; TextOff 'Exit'; PictureOff "ExitRuntime_KTP700_Basic_PN_TR"; PictureOn "ExitRuntime_KTP700_Basic_PN_TR"
      on Release: StopRuntime(0)
   Button "Template_Button" at 614,429 size 71x50; TextOff 'Text'
   Button "Template_Button_1" at 514,429 size 71x50; TextOff 'Text'
   Button "Template_Button_2" at 414,429 size 71x50; TextOff 'Text'
   Button "Template_Button_3" at 314,429 size 71x50; TextOff 'Text'
   Button "Template_Button_4" at 214,429 size 71x50; TextOff 'Text'
   Button "Template_Button_5" at 114,429 size 71x50; TextOff 'Text'
   Button "Start screen" at 14,429 size 71x50; TextOff 'Start screen'; PictureOff "NavigateHome_KTP700_Basic_PN_TR"; PictureOn "NavigateHome_KTP700_Basic_PN_TR"
      on Release: ActivateScreen("Screen_1", 0)

screen "Screen_1" 800x480
   GraphicView "Graphic view_1" at 0,0 size 799x480; Picture "600px-UK_Fin_Flash_low_visiability.svg"
   TextField "Text field_1" at 19,61 size 115x32; Text 'SENDING'
   TextField "Text field_2" at 256,61 size 138x32; Text 'RECEIVING'
   TextField "Text field_3" at 182,102 size 40x37; Text 'Hz'
   TextField "Text field_4" at 186,161 size 23x37; Text 'V'
   TextField "Text field_6" at 175,286 size 49x37; Text 'kW'
   TextField "Text field_7" at 179,352 size 39x37; Text 'PF'
   IOField "I/O field_1" at 31,99 size 100x40; FormatPattern 99999
      ProcessValue <- "Input_DB_Send_Frequency [Hz]"
   IOField "I/O field_2" at 30,161 size 100x40; FormatPattern 99999
      ProcessValue <- "Input_DB_Send_Voltage [V]"
   IOField "I/O field_3" at 29,286 size 100x40; FormatPattern 999999
      ProcessValue <- "Input_DB_Send_ActivePwr [W]"
   DateTimeField "Date/time field_1" at 588,456 size 211x24
   TextField "Text field_8" at 175,12 size 484x34; Text 'Power Distribution Monitoring System'
   Circle "Circle_1" at 419,75 size 66x66
      Appearance <- "Fault_DB_None"
   Circle "Circle_2" at 419,195 size 66x66
      Appearance <- "Fault_DB_Open_Circuit"
   Circle "Circle_3" at 558,71 size 66x66
      Appearance <- "Fault_DB_Low_Voltage"
   TextField "Text field_9" at 417,150 size 76x23; Text 'NORMAL'
   TextField "Text field_10" at 524,149 size 129x23; Text 'LOW VOLTAGE'
   TextField "Text field_11" at 400,263 size 131x23; Text 'OPEN CIRCUIT'
   Circle "Circle_4" at 558,197 size 66x66
      Appearance <- "Fault_DB_Short_Circuit"
   TextField "Text field_12" at 532,262 size 143x23; Text 'SHORT CIRCUIT'
   IOField "I/O field_4" at 29,223 size 100x40; FormatPattern 999999
      ProcessValue <- "Input_DB_Send_Current [mA]"
   IOField "I/O field_5" at 29,349 size 100x40; FormatPattern 99999
      ProcessValue <- "Input_DB_Send_PwrFactor"
   IOField "I/O field_6" at 276,99 size 100x40; FormatPattern 99999
      ProcessValue <- "Input_DB_Recv_Frequency [Hz]"
   IOField "I/O field_7" at 276,161 size 100x40; FormatPattern 99999
      ProcessValue <- "Input_DB_Recv_Voltage [V]"
   IOField "I/O field_8" at 275,223 size 100x40; FormatPattern 999999
      ProcessValue <- "Input_DB_Recv_Current [mA]"
   IOField "I/O field_9" at 275,286 size 100x40; FormatPattern 999999
      ProcessValue <- "Input_DB_Recv_ActivePwr [W]"
   IOField "I/O field_10" at 275,349 size 100x40; FormatPattern 99999
      ProcessValue <- "Input_DB_Recv_PwrFactor"
   Circle "Circle_5" at 419,297 size 66x66
      Appearance <- "Fault_DB_Illegal_Load"
   TextField "Text field_13" at 403,364 size 123x23; Text 'ILLEGAL LOAD'
   Circle "Circle_6" at 701,195 size 66x66
      Appearance <- "Fault_DB_Overload"
   TextField "Text field_14" at 688,261 size 95x23; Text 'OVERLOAD'
   Circle "Circle_7" at 558,297 size 66x66
      Appearance <- "Fault_DB_Poor_PF"
   TextField "Text field_15" at 558,365 size 77x23; Text 'POOR PF'
   Circle "Circle_8" at 701,71 size 66x66
      Appearance <- "Fault_DB_Freq_fault"
   TextField "Text field_16" at 677,149 size 109x23; Text 'FREQUENCY'
   TextField "Text field_5" at 189,223 size 23x37; Text 'A'
   Circle "Circle_9" at 142,66 size 27x27
      Appearance <- "Input_DB_Send_Error"
   Circle "Circle_10" at 228,66 size 27x27
      Appearance <- "Input_DB_Recv_Error"
   Switch "Switch_1" at 408,409 size 118x43; CaptionText 'Switch'; TextOff 'OFF'; TextOn 'ON'
      ProcessValue <- "Switch_manual"
      Visibility <- "Fault_DB_None"
   TextField "Text field_17" at 428,452 size 72x23; Text 'SWITCH'
*)

(* ===== HMI "HMI_RT_1" =====
system functions are stored by id; their names below are inferred from use
connection "Test_Conn": ETHERNET, SMART_S7_1200_OMS

HMI tags "Default tag table"
   "Fault_DB_Illegal_Load" : Bool = PLC Fault_DB.Illegal_Load, 1 s
   "Fault_DB_Low_Voltage" : Bool = PLC Fault_DB.Low_Voltage, 1 s
   "Fault_DB_Open_Circuit" : Bool = PLC Fault_DB.Open_Circuit, 1 s
   "Fault_DB_Overload" : Bool = PLC Fault_DB.Overload, 1 s
   "Fault_DB_Poor_PF" : Bool = PLC Fault_DB.Poor_PF, 1 s
   "Fault_DB_Short_Circuit" : Bool = PLC Fault_DB.Short_Circuit, 1 s
   "Input_DB_Recv_ActivePwr [W]" : DInt = PLC Input_DB."Recv_ActivePwr [W]", 1 s
   "Input_DB_Recv_Current [A]" : DInt = PLC Input_DB."Recv_Current [mA]", 1 s
   "Input_DB_Recv_Frequency [Hz]" : DInt = PLC Input_DB."Recv_Frequency [Hz]", 1 s
   "Input_DB_Recv_PwrFactor" : DInt = PLC Input_DB.Recv_PwrFactor, 1 s
   "Input_DB_Recv_Voltage [V]" : DInt = PLC Input_DB."Recv_Voltage [V]", 1 s
   "Input_DB_Send_ActivePwr [W]" : DInt = PLC Input_DB."Send_ActivePwr [W]", 1 s
   "Input_DB_Send_Current [A]" : DInt = PLC Input_DB."Send_Current [mA]", 1 s
   "Input_DB_Send_Energy [KWh]" : DInt = PLC Input_DB."Send_Energy [KWh]", 1 s
   "Input_DB_Send_Frequency [Hz]" : DInt = PLC Input_DB."Send_Frequency [Hz]", 1 s
   "Input_DB_Send_PwrFactor" : DInt = PLC Input_DB.Send_PwrFactor, 1 s
   "Input_DB_Send_Voltage [V]" : DInt = PLC Input_DB."Send_Voltage [V]", 1 s
   "Low_Volt" : Bool = PLC Low_Volt AT %M1.1, 1 s
   "Normal" : Bool = PLC Normal AT %M1.0, 1 s
   "Overload" : Bool = PLC Overload AT %M1.5, 1 s
   "Short_Circuit" : Bool = PLC Short_Circuit AT %M1.2, 1 s

screen "Screen_1" 800x480
   GraphicView "Graphic view_1" at 0,0 size 799x480; Picture "600px-UK_Fin_Flash_low_visiability.svg"
   TextField "Text field_1" at 39,59 size 115x32; Text 'SENDING'
   TextField "Text field_2" at 262,59 size 138x32; Text 'RECEIVING'
   TextField "Text field_3" at 191,111 size 40x37; Text 'Hz'
   TextField "Text field_4" at 185,173 size 73x37; Text 'Volts'
   TextField "Text field_5" at 168,234 size 106x37; Text 'mAmps'
   TextField "Text field_6" at 185,297 size 33x37; Text 'W'
   TextField "Text field_7" at 185,364 size 39x37; Text 'PF'
   IOField "I/O field_1" at 45,111 size 96x32; FormatPattern 9999
      ProcessValue <- "Input_DB_Send_Frequency [Hz]"
   IOField "I/O field_2" at 46,173 size 96x32; FormatPattern 99999
      ProcessValue <- "Input_DB_Send_Voltage [V]"
   IOField "I/O field_3" at 45,298 size 96x32; FormatPattern 99999
      ProcessValue <- "Input_DB_Send_ActivePwr [W]"
   DateTimeField "Date/time field_1" at 115,422 size 211x24
   TextField "Text field_8" at 175,12 size 484x34; Text 'Power Distribution Monitoring System'
   Circle "Circle_1" at 419,75 size 66x66
      Appearance <- "Normal"
   Circle "Circle_2" at 419,195 size 66x66
      Appearance <- "Fault_DB_Open_Circuit"
   Circle "Circle_3" at 558,71 size 66x66
      Appearance <- "Fault_DB_Low_Voltage"
   TextField "Text field_9" at 417,150 size 76x23; Text 'NORMAL'
   TextField "Text field_10" at 524,149 size 129x23; Text 'LOW VOLTAGE'
   TextField "Text field_11" at 400,263 size 131x23; Text 'OPEN CIRCUIT'
   Circle "Circle_4" at 558,197 size 66x66
      Appearance <- "Fault_DB_Short_Circuit"
   TextField "Text field_12" at 532,262 size 143x23; Text 'SHORT CIRCUIT'
   IOField "I/O field_4" at 45,235 size 96x32; FormatPattern 999
      ProcessValue <- "Input_DB_Send_Current [A]"
   IOField "I/O field_5" at 45,365 size 96x32; FormatPattern 999
      ProcessValue <- "Input_DB_Send_PwrFactor"
   IOField "I/O field_6" at 291,106 size 96x37; FormatPattern 999
      ProcessValue <- "Input_DB_Recv_Frequency [Hz]"
   IOField "I/O field_7" at 290,167 size 98x39; FormatPattern 99999
      ProcessValue <- "Input_DB_Recv_Voltage [V]"
   IOField "I/O field_8" at 289,233 size 98x39; FormatPattern 999
      ProcessValue <- "Input_DB_Recv_Current [A]"
   IOField "I/O field_9" at 290,300 size 97x38; FormatPattern 99999
      ProcessValue <- "Input_DB_Recv_ActivePwr [W]"
   IOField "I/O field_10" at 289,357 size 101x45; FormatPattern 999
      ProcessValue <- "Input_DB_Recv_PwrFactor"
   Circle "Circle_5" at 419,297 size 66x66
      Appearance <- "Fault_DB_Illegal_Load"
   TextField "Text field_13" at 403,364 size 123x23; Text 'ILLEGAL LOAD'
   Circle "Circle_6" at 701,195 size 66x66
      Appearance <- "Fault_DB_Overload"
   TextField "Text field_14" at 688,261 size 95x23; Text 'OVERLOAD'
   Circle "Circle_7" at 558,297 size 66x66
      Appearance <- "Fault_DB_Poor_PF"
   TextField "Text field_15" at 558,365 size 77x23; Text 'POOR PF'
   Circle "Circle_8" at 701,71 size 66x66
      Appearance <- "Short_Circuit"
   TextField "Text field_16" at 677,149 size 109x23; Text 'FREQUENCY'

Template "Template_1" 800x480
   Button "Exit" at 714,429 size 71x50; TextOn 'Exit'; TextOff 'Exit'; PictureOn "ExitRuntime_KTP700_Basic_PN_TR"; PictureOff "ExitRuntime_KTP700_Basic_PN_TR"
      on Release: StopRuntime(0)
   Button "Template_Button" at 614,429 size 71x50; TextOff 'Text'
   Button "Template_Button_1" at 514,429 size 71x50; TextOff 'Text'
   Button "Template_Button_2" at 414,429 size 71x50; TextOff 'Text'
   Button "Template_Button_3" at 314,429 size 71x50; TextOff 'Text'
   Button "Template_Button_4" at 214,429 size 71x50; TextOff 'Text'
   Button "Template_Button_5" at 114,429 size 71x50; TextOff 'Text'
   Button "Start screen" at 14,429 size 71x50; TextOn 'Start screen'; TextOff 'Start screen'; PictureOn "NavigateHome_KTP700_Basic_PN_TR"; PictureOff "NavigateHome_KTP700_Basic_PN_TR"
      on Release: ActivateScreen("Screen_1", 0)
*)

(* ===== HMI "PC_HMI" =====
connection "Main_PC": ETHERNET, S7_1200_OMS

HMI tags "Default tag table"
   "Fault_DB_Freq_fault" : Bool = PLC Fault_DB.Freq_fault, 1 s
   "Fault_DB_Illegal_Load" : Bool = PLC Fault_DB.Illegal_Load, 1 s
   "Fault_DB_Low_Voltage" : Bool = PLC Fault_DB.Low_Voltage, 1 s
   "Fault_DB_None" : Bool = PLC Fault_DB.None, 1 s
   "Fault_DB_Open_Circuit" : Bool = PLC Fault_DB.Open_Circuit, 1 s
   "Fault_DB_Overload" : Bool = PLC Fault_DB.Overload, 1 s
   "Fault_DB_Poor_PF" : Bool = PLC Fault_DB.Poor_PF, 1 s
   "Fault_DB_Short_Circuit" : Bool = PLC Fault_DB.Short_Circuit, 1 s
   "Input_DB_Recv_ActivePwr [W]" : DInt = PLC Input_DB."Recv_ActivePwr [W]", 1 s
   "Input_DB_Recv_Current [mA]" : DInt = PLC Input_DB."Recv_Current [A]", 1 s
   "Input_DB_Recv_Frequency [Hz]" : DInt = PLC Input_DB."Recv_Frequency [Hz]", 1 s
   "Input_DB_Recv_PwrFactor" : DInt = PLC Input_DB.Recv_PwrFactor, 1 s
   "Input_DB_Recv_Voltage [V]" : DInt = PLC Input_DB."Recv_Voltage [V]", 1 s
   "Input_DB_Send_ActivePwr [W]" : DInt = PLC Input_DB."Send_ActivePwr [W]", 1 s
   "Input_DB_Send_Current [mA]" : DInt = PLC Input_DB."Send_Current [A]", 1 s
   "Input_DB_Send_Frequency [Hz]" : DInt = PLC Input_DB."Send_Frequency [Hz]", 1 s
   "Input_DB_Send_PwrFactor" : DInt = PLC Input_DB.Send_PwrFactor, 1 s
   "Input_DB_Send_Voltage [V]" : DInt = PLC Input_DB."Send_Voltage [V]", 1 s

screen "Screen_1" 1024x768
   GraphicView "Graphic view_1" at 0,0 size 799x480; Picture "600px-UK_Fin_Flash_low_visiability.svg"
   TextField "Text field_1" at 39,59 size 115x32; Text 'SENDING'
   TextField "Text field_2" at 262,59 size 138x32; Text 'RECEIVING'
   TextField "Text field_3" at 191,111 size 40x37; Text 'Hz'
   TextField "Text field_4" at 185,173 size 73x37; Text 'Volts'
   TextField "Text field_5" at 168,234 size 106x37; Text 'mAmps'
   TextField "Text field_6" at 185,297 size 33x37; Text 'W'
   TextField "Text field_7" at 185,364 size 39x37; Text 'PF'
   IOField "I/O field_1" at 45,111 size 96x32; FormatPattern 9999
      ProcessValue <- "Input_DB_Send_Frequency [Hz]"
   IOField "I/O field_2" at 46,173 size 96x32; FormatPattern 99999
      ProcessValue <- "Input_DB_Send_Voltage [V]"
   IOField "I/O field_3" at 45,298 size 96x32; FormatPattern 99999
      ProcessValue <- "Input_DB_Send_ActivePwr [W]"
   DateTimeField "Date/time field_1" at 115,422 size 211x24
   TextField "Text field_8" at 175,12 size 484x34; Text 'Power Distribution Monitoring System'
   Circle "Circle_1" at 419,75 size 66x66
      Appearance <- "Fault_DB_None"
   Circle "Circle_2" at 419,195 size 66x66
      Appearance <- "Fault_DB_Open_Circuit"
   Circle "Circle_3" at 558,71 size 66x66
      Appearance <- "Fault_DB_Low_Voltage"
   TextField "Text field_9" at 417,150 size 76x23; Text 'NORMAL'
   TextField "Text field_10" at 524,149 size 129x23; Text 'LOW VOLTAGE'
   TextField "Text field_11" at 400,263 size 131x23; Text 'OPEN CIRCUIT'
   Circle "Circle_4" at 558,197 size 66x66
      Appearance <- "Fault_DB_Short_Circuit"
   TextField "Text field_12" at 532,262 size 143x23; Text 'SHORT CIRCUIT'
   IOField "I/O field_4" at 45,235 size 96x32; FormatPattern 999
      ProcessValue <- "Input_DB_Send_Current [mA]"
   IOField "I/O field_5" at 45,365 size 96x32; FormatPattern 999
      ProcessValue <- "Input_DB_Send_PwrFactor"
   IOField "I/O field_6" at 291,106 size 96x37; FormatPattern 999
      ProcessValue <- "Input_DB_Recv_Frequency [Hz]"
   IOField "I/O field_7" at 290,167 size 98x39; FormatPattern 99999
      ProcessValue <- "Input_DB_Recv_Voltage [V]"
   IOField "I/O field_8" at 289,233 size 98x39; FormatPattern 999
      ProcessValue <- "Input_DB_Recv_Current [mA]"
   IOField "I/O field_9" at 290,300 size 97x38; FormatPattern 99999
      ProcessValue <- "Input_DB_Recv_ActivePwr [W]"
   IOField "I/O field_10" at 289,357 size 101x45; FormatPattern 999
      ProcessValue <- "Input_DB_Recv_PwrFactor"
   Circle "Circle_5" at 419,297 size 66x66
      Appearance <- "Fault_DB_Illegal_Load"
   TextField "Text field_13" at 403,364 size 123x23; Text 'ILLEGAL LOAD'
   Circle "Circle_6" at 701,195 size 66x66
      Appearance <- "Fault_DB_Overload"
   TextField "Text field_14" at 688,261 size 95x23; Text 'OVERLOAD'
   Circle "Circle_7" at 558,297 size 66x66
      Appearance <- "Fault_DB_Poor_PF"
   TextField "Text field_15" at 558,365 size 77x23; Text 'POOR PF'
   Circle "Circle_8" at 701,71 size 66x66
      Appearance <- "Fault_DB_Freq_fault"
   TextField "Text field_16" at 677,149 size 109x23; Text 'FREQUENCY'
*)